RoboDK station: Tarea3_IsabellaCeballos.rdk

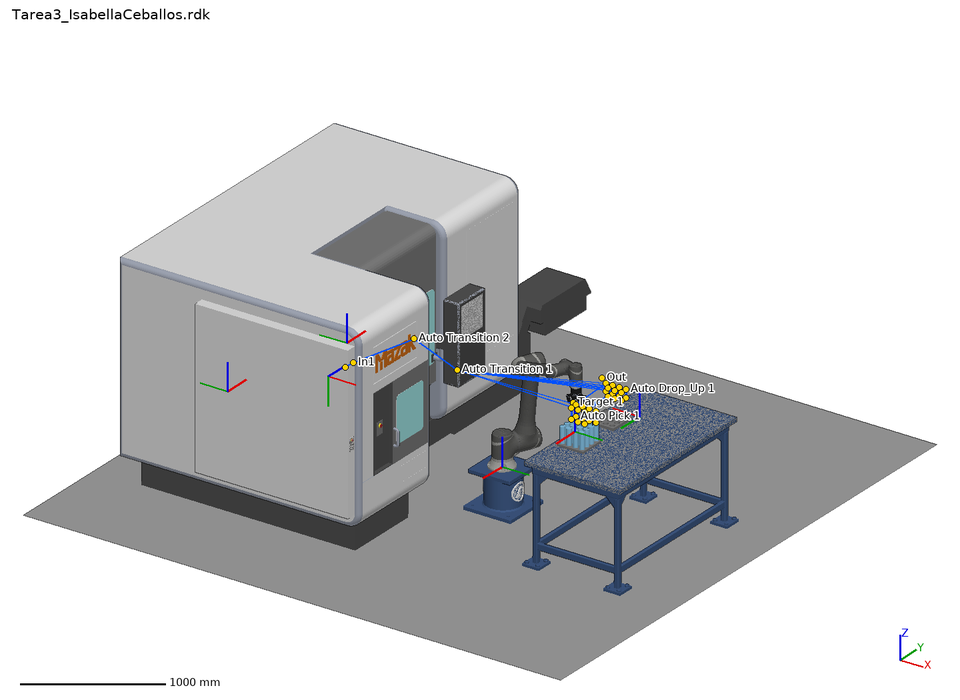
[picture v0: the station drawn from its stored meshes, robots at their saved joint values, targets as dots, program paths as lines]
Station Tarea3_IsabellaCeballos (saved by RoboDK 5.6.0). Poses are relative to the parent item; angles as X-Y-Z fixed-axis rotations.
Station parameters (name, value as stored): TAGS, ['Machine Tending', 'CNC']
  - frame Omron TM12X Base at (300, 0, 70) mm, rotated rx 0 ry 0 rz -90 deg
    - robot Omron TM12X: 6 axes, payload 12 kg, reach 1300 mm, repeatability 0.1 mm, weight 33.3 kg
        modified DH rows (alpha deg, a mm, theta deg, d mm): 0, 0, 0, 165.2; 90, 0, 90, 0; 0, 636.1, 0, 0; 0, 557.9, -90, 156.3; -90, 0, 0, 106; 90, 0, 180, 113.15
        joint limits [-360, -360, -163, -360, -360, -360] to [360, 360, 163, 360, 360, 360]; home [0, 0, 90, -90, 90, 0]; saved at [245.421, -8.702, -61.622, -16.467, -90.498, 224.904]
      - tool g1, TCP at (0, 0, 130) mm, size 134.4 x 157.6 x 75 mm
      - tool RobotiQ 2F-85 Gripper (Open), TCP at (0, 0, 130) mm, size 147.4 x 146.8 x 75 mm
    - object Pedestal H12in (Type 1) at (0, 10, -300) mm, size 400 x 400 x 304.8 mm, geometry from Pedestal-H12in-Type-1.sld
  - frame Mazak Lathe Base at (-1000, 0, 650) mm, rotated rx 0 ry 0 rz 90 deg
    - robot Mazak Lathe: 1 axes
        modified DH rows (alpha deg, a mm, theta deg, d mm): 0, 0, 0, 0 linear
        base shift (0, 0, 0) mm, rotated rx 0 ry 90 rz 0 deg
        joint limits [0] to [700]; home [0]; saved at [0]
    - frame Lathe at (-368.68, -104.77, -79.13) mm, rotated rx -90 ry 0 rz -90 deg
  - frame Input at (1010, -140, 590) mm, rotated rx 0 ry 0 rz -90 deg
    - object Part Matrix at (0, 0, 0) mm, size 220 x 220 x 25 mm, geometry from Part Matrix.step
    - target Target 1 (Cartesian target) at (-26.53, -36.52, 202.61) mm, rotated rx -177.37 ry 1.91 rz -69.45 deg; joints [247.43, -1, -72.52, -13.29, -90.61, 226.91] of Omron TM12X
    - object Part 8 at (137.5, 27.5, -20) mm, size 40 x 40 x 150 mm, geometry from Part.step
    - object Part 6 at (137.5, 137.5, -20) mm, size 40 x 40 x 150 mm, geometry from Part.step
    - object Part 1 at (192.5, 192.5, -20) mm, size 40 x 40 x 150 mm, geometry from Part.step
    - object Part 5 at (137.5, 192.5, -20) mm, size 40 x 40 x 150 mm, geometry from Part.step
    - object Part 7 at (137.5, 82.5, -20) mm, size 40 x 40 x 150 mm, geometry from Part.step
    - object Part 4 at (192.5, 27.5, -20) mm, rotated rx 0 ry 0 rz -180 deg, size 40 x 40 x 150 mm, geometry from Part.step
    - object Part 3 at (192.5, 82.5, -20) mm, rotated rx 0 ry 0 rz -180 deg, size 40 x 40 x 150 mm, geometry from Part.step
    - object Part 2 at (192.5, 137.5, -20) mm, rotated rx 0 ry 0 rz -180 deg, size 40 x 40 x 150 mm, geometry from Part.step
    - target Home (Cartesian target) at (28, 28, 225) mm, rotated rx -177.37 ry 1.91 rz -69.45 deg; joints [245.421, -8.702, -61.622, -16.467, -90.498, 224.904] of Omron TM12X
    - target Out (Cartesian target) at (-374.96, -36.47, 250.91) mm, rotated rx 179.32 ry 1.81 rz -82.53 deg; joints [276.325, -63.11, 61.627, -86.724, -89.287, -91.145] of Omron TM12X
    - object Part 14 at (27.5, 137.5, -20) mm, size 40 x 40 x 150 mm, geometry from Part.step
    - object Part 13 at (27.5, 192.5, -20) mm, size 40 x 40 x 150 mm, geometry from Part.step
    - object Part 11 at (82.5, 82.5, -20) mm, size 40 x 40 x 150 mm, geometry from Part.step
    - object Part 10 at (82.5, 137.5, -20) mm, size 40 x 40 x 150 mm, geometry from Part.step
    - object Part 9 at (82.5, 192.5, -20) mm, size 40 x 40 x 150 mm, geometry from Part.step
    - object Part 12 at (82.5, 27.5, -20) mm, size 40 x 40 x 150 mm, geometry from Part.step
    - object Part 15 at (27.5, 82.5, -20) mm, size 40 x 40 x 150 mm, geometry from Part.step
    - object Part 16 at (27.5, 27.5, -20) mm, size 40 x 40 x 150 mm, geometry from Part.step
    - target Auto Transition 1 (Cartesian target) at (259.07, -803.97, 350.52) mm, rotated rx -177.37 ry 1.91 rz -69.45 deg; joints [142.248, 16.086, -68.881, -37.451, -86.762, 121.738] of Omron TM12X
    - target Auto Transition 2 (Cartesian target) at (28.12, -1329.27, 350.52) mm, rotated rx -177.37 ry 1.91 rz -69.45 deg; joints [90.384, -51.512, 48.629, -89.818, -88.195, 69.839] of Omron TM12X
    - target Auto Up_Pick 1 (Cartesian target) at (28, 28, 225) mm, rotated rx -177.37 ry 1.91 rz -69.45 deg; joints [245.421, -8.702, -61.622, -16.467, -90.498, 224.904] of Omron TM12X
    - target Auto Pick 1 (Cartesian target) at (28, 28, 135) mm, rotated rx -177.37 ry 1.91 rz -69.45 deg; joints [245.421, -6.476, -73.764, -6.551, -90.498, 224.904] of Omron TM12X
    - target Auto Drop_Up 1 (Cartesian target) at (-374.01, 165.11, 220.31) mm, rotated rx -177.37 ry 1.91 rz -69.45 deg; joints [275.591, -25.399, -39.284, -22.792, -92.043, 255.043] of Omron TM12X
    - target Auto Drop 1 (Cartesian target) at (-374.01, 165.11, 156.87) mm, rotated rx -177.37 ry 1.91 rz -69.45 deg; joints [275.591, -22.487, -50.629, -14.358, -92.043, 255.043] of Omron TM12X
    - target Auto Up_Pick 2 (Cartesian target) at (28, 84, 225) mm, rotated rx -177.37 ry 1.91 rz -69.45 deg; joints [247.13, -14.265, -54.709, -17.833, -90.593, 226.611] of Omron TM12X
    - target Auto Pick 2 (Cartesian target) at (28, 84, 135) mm, rotated rx -177.37 ry 1.91 rz -69.45 deg; joints [247.13, -11.733, -67.54, -7.534, -90.593, 226.611] of Omron TM12X
    - target Auto Drop_Up 2 (Cartesian target) at (-374.01, 109.11, 220.31) mm, rotated rx -177.37 ry 1.91 rz -69.45 deg; joints [275.969, -18.914, -48.812, -19.762, -92.059, 255.421] of Omron TM12X
    - target Auto Drop 2 (Cartesian target) at (-374.01, 109.11, 156.87) mm, rotated rx -177.37 ry 1.91 rz -69.45 deg; joints [275.969, -16.675, -58.745, -12.068, -92.059, 255.421] of Omron TM12X
    - target Auto Up_Pick 3 (Cartesian target) at (28, 140, 225) mm, rotated rx -177.37 ry 1.91 rz -69.45 deg; joints [248.62, -20.312, -46.448, -20.064, -90.676, 228.098] of Omron TM12X
    - target Auto Pick 3 (Cartesian target) at (28, 140, 135) mm, rotated rx -177.37 ry 1.91 rz -69.45 deg; joints [248.62, -17.229, -60.442, -9.153, -90.676, 228.098] of Omron TM12X
    - target Auto Drop_Up 3 (Cartesian target) at (-374.01, 53.11, 220.31) mm, rotated rx -177.37 ry 1.91 rz -69.45 deg; joints [276.4, -13.16, -56.507, -17.837, -92.078, 255.852] of Omron TM12X
    - target Auto Drop 3 (Cartesian target) at (-374.01, 53.11, 156.87) mm, rotated rx -177.37 ry 1.91 rz -69.45 deg; joints [276.4, -11.285, -65.66, -10.558, -92.078, 255.852] of Omron TM12X
    - target Auto Up_Pick 4 (Cartesian target) at (28, 196, 225) mm, rotated rx -177.37 ry 1.91 rz -69.45 deg; joints [249.929, -27.249, -35.99, -23.601, -90.748, 229.406] of Omron TM12X
    - target Auto Pick 4 (Cartesian target) at (28, 196, 135) mm, rotated rx -177.37 ry 1.91 rz -69.45 deg; joints [249.929, -23.122, -52.163, -11.554, -90.748, 229.406] of Omron TM12X
    - target Auto Drop_Up 4 (Cartesian target) at (-374.01, -2.89, 220.31) mm, rotated rx -177.37 ry 1.91 rz -69.45 deg; joints [276.898, -7.834, -63.005, -16.683, -92.1, 256.35] of Omron TM12X
    - target Auto Drop 4 (Cartesian target) at (-374.01, -2.89, 156.87) mm, rotated rx -177.37 ry 1.91 rz -69.45 deg; joints [276.898, -6.163, -71.686, -9.672, -92.1, 256.35] of Omron TM12X
    - target Auto Up_Pick 5 (Cartesian target) at (84, 28, 225) mm, rotated rx -177.37 ry 1.91 rz -69.45 deg; joints [241.513, -10.095, -59.958, -16.711, -90.278, 221.002] of Omron TM12X
    - target Auto Pick 5 (Cartesian target) at (84, 28, 135) mm, rotated rx -177.37 ry 1.91 rz -69.45 deg; joints [241.513, -7.808, -72.245, -6.712, -90.278, 221.002] of Omron TM12X
    - target Auto Drop_Up 5 (Cartesian target) at (-318.01, 165.11, 220.31) mm, rotated rx -177.37 ry 1.91 rz -69.45 deg; joints [271.937, -23.672, -41.937, -21.74, -91.878, 251.39] of Omron TM12X
    - target Auto Drop 5 (Cartesian target) at (-318.01, 165.11, 156.87) mm, rotated rx -177.37 ry 1.91 rz -69.45 deg; joints [271.937, -20.979, -52.826, -13.544, -91.878, 251.39] of Omron TM12X
    - target Auto Up_Pick 6 (Cartesian target) at (84, 84, 225) mm, rotated rx -177.37 ry 1.91 rz -69.45 deg; joints [243.44, -15.653, -52.889, -18.233, -90.387, 222.926] of Omron TM12X
    - target Auto Pick 6 (Cartesian target) at (84, 84, 135) mm, rotated rx -177.37 ry 1.91 rz -69.45 deg; joints [243.44, -13.018, -65.941, -7.816, -90.387, 222.926] of Omron TM12X
    - target Auto Drop_Up 6 (Cartesian target) at (-318.01, 109.11, 220.31) mm, rotated rx -177.37 ry 1.91 rz -69.45 deg; joints [272.07, -17.314, -51.051, -18.989, -91.884, 251.524] of Omron TM12X
    - target Auto Drop 6 (Cartesian target) at (-318.01, 109.11, 156.87) mm, rotated rx -177.37 ry 1.91 rz -69.45 deg; joints [272.07, -15.198, -60.726, -11.43, -91.884, 251.524] of Omron TM12X
    - target Auto Up_Pick 7 (Cartesian target) at (84, 140, 225) mm, rotated rx -177.37 ry 1.91 rz -69.45 deg; joints [245.13, -21.756, -44.367, -20.666, -90.482, 224.613] of Omron TM12X
    - target Auto Pick 7 (Cartesian target) at (84, 140, 135) mm, rotated rx -177.37 ry 1.91 rz -69.45 deg; joints [245.13, -18.5, -58.722, -9.566, -90.482, 224.613] of Omron TM12X
    - target Auto Drop_Up 7 (Cartesian target) at (-318.01, 53.11, 220.31) mm, rotated rx -177.37 ry 1.91 rz -69.45 deg; joints [272.223, -11.586, -58.52, -17.253, -91.891, 251.676] of Omron TM12X
    - target Auto Drop 7 (Cartesian target) at (-318.01, 53.11, 156.87) mm, rotated rx -177.37 ry 1.91 rz -69.45 deg; joints [272.223, -9.786, -67.508, -10.065, -91.891, 251.676] of Omron TM12X
  - frame Output at (1250, 290, 600) mm, rotated rx 0 ry 0 rz -180 deg
    - object Part Matrix at (47.8, 28.1, 0) mm, size 220 x 220 x 25 mm, geometry from Part Matrix.step
  - frame World at (-2000, 0, 0) mm, rotated rx 0 ry 0 rz 90 deg
    - object Floor at (250, -1940, -230) mm, size 4500 x 4500 x 0 mm, geometry from Floor (2).sld
    - object Table 1400x800x800mm at (-340, -3360, 570) mm, size 1420 x 820 x 800 mm, geometry from Table-1400x800x800mm.sld
    - target OpenDoor (Cartesian target) at (700, -1000, 650) mm; joints [700] of Mazak Lathe
    - target CloseDoor (Cartesian target) at (0, -1000, 650) mm; joints [0] of Mazak Lathe
    - target In1 (Cartesian target) at (-137.95, -1150.25, 595.88) mm, rotated rx -86.34 ry 2.11 rz 94.34 deg; joints [77.244, -89.992, 25.646, 51.981, -342.661, 170.292] of Omron TM12X
    - target In2 (Cartesian target) at (-206.56, -1130.76, 584.67) mm, rotated rx -87.8 ry 7.87 rz 92.76 deg; joints [-84.147, 66.082, 6.025, 75.079, -175.968, 40.623] of Omron TM12X
  - Python program pick_Up (listed below)
  - program atach (1 instructions, listed below)
  - program detach (1 instructions, listed below)
  - program init (1 instructions, listed below)
  - program OpenDoor (2 instructions, listed below)
  - program CloseDoor (2 instructions, listed below)
  - program GoHome (3 instructions, listed below)
  - program Go_Out (3 instructions, listed below)
  - program Main_Program (214 instructions, listed below)
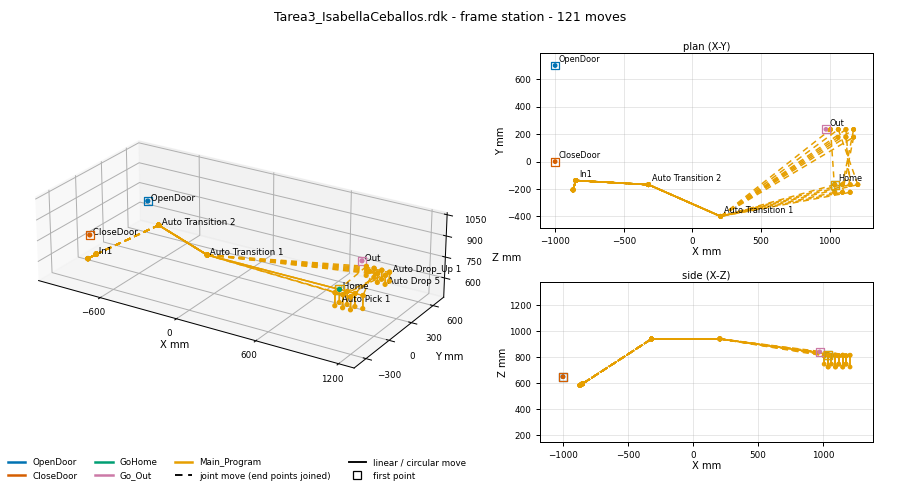
[picture p0: tool path of Tarea3_IsabellaCeballos.rdk in frame station, 121 of 121 moves have a stored position in this frame; points joined in program order, loops and branches not executed]

--- Python program pick_Up ---
import tkinter as tk
import time as t
from robolink import *    # Robot toolbox



# Link to RoboDK
RDK = Robolink() # Interactuar con la interfaz del robot

# Mecanismos
robot = RDK.Item("Omron TM12X", ITEM_TYPE_ROBOT) #Robot
MAZAK = RDK.Item("Mazak Lathe") # Mazak
Tool_gripper = RDK.Item('g1',ITEM_TYPE_TOOL ) #Gripper

#Esto es para que no se repitan cosas en el código
list_names = RDK.ItemList(None, True)
for item_name in list_names:
    if item_name.startswith('Auto'):
        RDK.Item(item_name).Delete()
    if item_name.startswith('Main_'):
        RDK.Item(item_name).Delete()

#Código para generar puntos de botellas
def gridXY (m,n,d, e):

    """
     m= número de puntos en x
     n= número de puntos en y
     d= distancia entre cada punto en m

     En este ejercicio m = n, es cuadrado el soporte. 4x4
    """

    lista_puntos = []
    coeficientes = [1, 3, 5, 7 ]
    for i in range(m):
        for j in range(n):
            punto = [coeficientes[i]*d, coeficientes[j]*e, 225.000]
            lista_puntos.append(punto)


    return lista_puntos

m = 4
n = 4
d = 28
e = 28


puntos = gridXY(m,n,d,e)


# Código Principal

# Marcos de referencias
Input = RDK.Item("Input",ITEM_TYPE_FRAME) #frame
Output = RDK.Item("Output",ITEM_TYPE_FRAME)#frame2
Lathe = RDK.Item("Lathe",ITEM_TYPE_FRAME) #frame3
World = RDK.Item("World",ITEM_TYPE_FRAME) #frame4



robot.setPoseFrame(Input) #asociamos el robot a Input
pose_ref = robot.Pose()

Program = RDK.AddProgram('Main_Program')# Se genera programa


j = 0

#TARGETS DEL PROGRAMA

In1 = RDK.Item('In1',ITEM_TYPE_TARGET)
In2 = RDK.Item('In2',ITEM_TYPE_TARGET)
In3 = RDK.Item('In3',ITEM_TYPE_TARGET)


robot.setPoseFrame(Input)

    #TRANSITION 1
Trans1 = RDK.AddTarget('Auto Transition 1')#ti7
pose_t = pose_ref
pose_t.setPos([259.072, -803.965, 350.521] )
Trans1.setPose(pose_t)
Trans1.setAsCartesianTarget()
Trans1.setVisible(0)

    #TRANSITION 2
Trans2 = RDK.AddTarget('Auto Transition 2') #ti9
pose_t.setPos([28.119, -1329.271, 350.521] )
Trans2.setPose(pose_t)
Trans2.setAsCartesianTarget()
Trans2.setVisible(0)

# Funciones del programa

def Pick_up(P,Pick_Up,Pick):
    P.MoveJ(Pick_Up)
    t.sleep(0.5)
    P.MoveL(Pick)
    t.sleep(0.5)
    P.RunInstruction('atach',0)
    t.sleep(0.5)
    P.MoveL(Pick_Up)
    t.sleep(0.5)
    return

def Drop_out(P,Drop,Drop_Up):
    P.MoveJ(Drop_Up)
    t.sleep(0.5)
    P.MoveL(Drop)
    t.sleep(0.5)
    P.RunInstruction('detach',0)
    t.sleep(0.5)
    P.MoveL(Drop_Up)
    t.sleep(0.5)
    return

def Pick_Lathe_Transition(P,Trans1,Trans2):
    P.MoveJ(Trans1)
    t.sleep(0.5)
    P.MoveJ(Trans2)
    t.sleep(0.5)
    return

def PickLathe(P,In1,In2,In3,Trans2):
    P.setFrame(World)
    P.MoveJ(In1)
    P.MoveL(In2)
    P.RunInstruction('detach',0)
    t.sleep(0.5)
    P.MoveL(In1)
    t.sleep(0.5)
    P.setFrame(Input)
    t.sleep(0.5)
    P.MoveJ(Trans2)
    t.sleep(5)
    return

def DropLathe(P,In1,In2,Trans2):
    P.setFrame(World)
    P.MoveJ(In1)
    P.MoveL(In2)
    P.RunInstruction('atach',0)
    t.sleep(0.5)
    P.MoveL(In1)
    t.sleep(0.5)
    P.setFrame(Input)
    t.sleep(0.5)
    P.MoveJ(Trans2)
    t.sleep(5)
    return


for i in puntos:

    #**GENARACIÓN DE TARGETS PICK BOTELLAS**
    #---------------------------------------
    robot.setPoseFrame(Input)
    Pick_Up = RDK.AddTarget('Auto Up_Pick %i' %(j+1))
    pose_i = pose_ref
    pose_i.setPos(i) #lista [x,y,z]
    Pick_Up.setPose(pose_i)
    Pick_Up.setAsCartesianTarget()
    Pick_Up.setVisible(0)
    #--------------------------------------
    Pick = RDK.AddTarget('Auto Pick %i' %(j+1))
    pose_j = pose_i
    pose_j.setPos([i[0],i[1], 135] )#[x,y,z]
    Pick.setPose(pose_j)
    Pick.setAsCartesianTarget()
    Pick.setVisible(0)



    #**GENERACIÓN DE TARGETS DROP BOTELLAS**
    #---------------------------------------
    Drop_Up = RDK.AddTarget('Auto Drop_Up %i' %(j+1))
    pose_p = pose_i
    pose_p.setPos([-402.010 + i[0], 193.114 - i[1], 220.306] )#[x,y,z]
    Drop_Up.setPose(pose_p)
    Drop_Up.setAsCartesianTarget()
    Drop_Up.setVisible(0)
   #---------------------------------------
    Drop = RDK.AddTarget('Auto Drop %i' %(j+1))
    pose_r = pose_i
    pose_r.setPos([-402.010 + i[0], 193.114 - i[1], 156.874] )#[x,y,z]
    Drop.setPose(pose_r)
    Drop.setAsCartesianTarget()
    Drop.setVisible(0)



    # SECUENCIA
    Program.setFrame(Input)
    Pick_up(Program,Pick_Up,Pick)
    Pick_Lathe_Transition(Program,Trans1,Trans2)
    Program.RunInstruction('OpenDoor',0)
    PickLathe(Program,In1,In2,In3,Trans2)
    Program.RunInstruction('CloseDoor',0)
    Program.RunInstruction('OpenDoor',0)
    DropLathe(Program,In1,In2,Trans2)
    Program.RunInstruction('CloseDoor',0)
    Program.MoveL(Trans1)
    Program.RunInstruction('Go_Out',0)
    Drop_out(Program,Drop,Drop_Up)


    j+=1

--- program atach (robot Omron TM12X) ---
  Adjuntar a g1

--- program detach (robot Omron TM12X) ---
  Separar de g1

--- program init (robot Omron TM12X) ---
  Reemplazar objetos

--- program OpenDoor (robot Mazak Lathe) ---
  Est. Ref.: World
  MoveJ (OpenDoor)

--- program CloseDoor (robot Mazak Lathe) ---
  Est. Ref.: World
  MoveJ (CloseDoor)

--- program GoHome (robot Omron TM12X) ---
  Est. Ref.: Input
  Est. herr: g1
  MoveJ (Home)

--- program Go_Out (robot Omron TM12X) ---
  Est. Ref.: Input
  Est. herr: g1
  MoveJ (Out)

--- program Main_Program (robot Omron TM12X) ---
  Set Ref.: Input
  MoveJ (Auto Up_Pick 1)
  MoveL (Auto Pick 1)
  Call atach
  MoveL (Auto Up_Pick 1)
  MoveJ (Auto Transition 1)
  MoveJ (Auto Transition 2)
  Call OpenDoor
  Set Ref.: World
  MoveJ (In1)
  MoveL (In2)
  Call detach
  MoveL (In1)
  Set Ref.: Input
  MoveJ (Auto Transition 2)
  Call CloseDoor
  Call OpenDoor
  Set Ref.: World
  MoveJ (In1)
  MoveL (In2)
  Call atach
  MoveL (In1)
  Set Ref.: Input
  MoveJ (Auto Transition 2)
  Call CloseDoor
  MoveL (Auto Transition 1)
  Call Go_Out
  MoveJ (Auto Drop_Up 1)
  MoveL (Auto Drop 1)
  Call detach
  MoveL (Auto Drop_Up 1)
  Set Ref.: Input
  MoveJ (Auto Up_Pick 2)
  MoveL (Auto Pick 2)
  Call atach
  MoveL (Auto Up_Pick 2)
  MoveJ (Auto Transition 1)
  MoveJ (Auto Transition 2)
  Call OpenDoor
  Set Ref.: World
  MoveJ (In1)
  MoveL (In2)
  Call detach
  MoveL (In1)
  Set Ref.: Input
  MoveJ (Auto Transition 2)
  Call CloseDoor
  Call OpenDoor
  Set Ref.: World
  MoveJ (In1)
  MoveL (In2)
  Call atach
  MoveL (In1)
  Set Ref.: Input
  MoveJ (Auto Transition 2)
  Call CloseDoor
  MoveL (Auto Transition 1)
  Call Go_Out
  MoveJ (Auto Drop_Up 2)
  MoveL (Auto Drop 2)
  Call detach
  MoveL (Auto Drop_Up 2)
  Set Ref.: Input
  MoveJ (Auto Up_Pick 3)
  MoveL (Auto Pick 3)
  Call atach
  MoveL (Auto Up_Pick 3)
  MoveJ (Auto Transition 1)
  MoveJ (Auto Transition 2)
  Call OpenDoor
  Set Ref.: World
  MoveJ (In1)
  MoveL (In2)
  Call detach
  MoveL (In1)
  Set Ref.: Input
  MoveJ (Auto Transition 2)
  Call CloseDoor
  Call OpenDoor
  Set Ref.: World
  MoveJ (In1)
  MoveL (In2)
  Call atach
  MoveL (In1)
  Set Ref.: Input
  MoveJ (Auto Transition 2)
  Call CloseDoor
  MoveL (Auto Transition 1)
  Call Go_Out
  MoveJ (Auto Drop_Up 3)
  MoveL (Auto Drop 3)
  Call detach
  MoveL (Auto Drop_Up 3)
  Set Ref.: Input
  MoveJ (Auto Up_Pick 4)
  MoveL (Auto Pick 4)
  Call atach
  MoveL (Auto Up_Pick 4)
  MoveJ (Auto Transition 1)
  MoveJ (Auto Transition 2)
  Call OpenDoor
  Set Ref.: World
  MoveJ (In1)
  MoveL (In2)
  Call detach
  MoveL (In1)
  Set Ref.: Input
  MoveJ (Auto Transition 2)
  Call CloseDoor
  Call OpenDoor
  Set Ref.: World
  MoveJ (In1)
  MoveL (In2)
  Call atach
  MoveL (In1)
  Set Ref.: Input
  MoveJ (Auto Transition 2)
  Call CloseDoor
  MoveL (Auto Transition 1)
  Call Go_Out
  MoveJ (Auto Drop_Up 4)
  MoveL (Auto Drop 4)
  Call detach
  MoveL (Auto Drop_Up 4)
  Set Ref.: Input
  MoveJ (Auto Up_Pick 5)
  MoveL (Auto Pick 5)
  Call atach
  MoveL (Auto Up_Pick 5)
  MoveJ (Auto Transition 1)
  MoveJ (Auto Transition 2)
  Call OpenDoor
  Set Ref.: World
  MoveJ (In1)
  MoveL (In2)
  Call detach
  MoveL (In1)
  Set Ref.: Input
  MoveJ (Auto Transition 2)
  Call CloseDoor
  Call OpenDoor
  Set Ref.: World
  MoveJ (In1)
  MoveL (In2)
  Call atach
  MoveL (In1)
  Set Ref.: Input
  MoveJ (Auto Transition 2)
  Call CloseDoor
  MoveL (Auto Transition 1)
  Call Go_Out
  MoveJ (Auto Drop_Up 5)
  MoveL (Auto Drop 5)
  Call detach
  MoveL (Auto Drop_Up 5)
  Set Ref.: Input
  MoveJ (Auto Up_Pick 6)
  MoveL (Auto Pick 6)
  Call atach
  MoveL (Auto Up_Pick 6)
  MoveJ (Auto Transition 1)
  MoveJ (Auto Transition 2)
  Call OpenDoor
  Set Ref.: World
  MoveJ (In1)
  MoveL (In2)
  Call detach
  MoveL (In1)
  Set Ref.: Input
  MoveJ (Auto Transition 2)
  Call CloseDoor
  Call OpenDoor
  Set Ref.: World
  MoveJ (In1)
  MoveL (In2)
  Call atach
  MoveL (In1)
  Set Ref.: Input
  MoveJ (Auto Transition 2)
  Call CloseDoor
  MoveL (Auto Transition 1)
  Call Go_Out
  MoveJ (Auto Drop_Up 6)
  MoveL (Auto Drop 6)
  Call detach
  MoveL (Auto Drop_Up 6)
  Set Ref.: Input
  MoveJ (Auto Up_Pick 7)
  MoveL (Auto Pick 7)
  Call atach
  MoveL (Auto Up_Pick 7)
  MoveJ (Auto Transition 1)
  MoveJ (Auto Transition 2)
  Call OpenDoor
  Set Ref.: World
  MoveJ (In1)
  MoveL (In2)
  Call detach
  MoveL (In1)
  Set Ref.: Input
  MoveJ (Auto Transition 2)
  Call CloseDoor
  Call OpenDoor
  Set Ref.: World
  MoveJ (In1)
  MoveL (In2)
  Call atach
  MoveL (In1)
  Set Ref.: Input
  MoveJ (Auto Transition 2)
  Call CloseDoor
  MoveL (Auto Transition 1)
  Call Go_Out
  MoveJ (Auto Drop_Up 7)
